				//Oś 1 staneła
				IF bRun1 AND ABS(Screwing1AxisRef.NcToPlc.ActVelo) < 150 THEN  //bylo 300
					mcHeightGearInMultiMaster.GearRatio1 	:=	0;
					mcHeightGearInMultiMaster.GearRatio2 	:=	lrSf2 * 	lrGearRatio2;
				END_IF
				//Oś 2 staneła		
				IF bRun2 AND ABS(Screwing2AxisRef.NcToPlc.ActVelo) < 150 THEN //bylo 300
					mcHeightGearInMultiMaster.GearRatio1 	:=	lrSf1 * 	lrGearRatio1;	
					mcHeightGearInMultiMaster.GearRatio2 	:=	0;				
				END_IF
				//Całkowite zatrzymanie - dwie osie staneły
				IF ABS(Screwing1AxisRef.NcToPlc.ActVelo) < 150 AND ABS(Screwing2AxisRef.NcToPlc.ActVelo) < 150 THEN //bylo 300
					mcHeightGearInMultiMaster.GearRatio1 	:=	0;
					mcHeightGearInMultiMaster.GearRatio2 	:=	0;	
				END_IF
				
				IF NOT bOptionMomentaryMode THEN	
					Running6ScrewingPositionTorqueMode();
				ELSE
					Running6ScrewingMomentaryMode();								
				END_IF
			END_IF
//====================================

	(*Przytrzymanie / Czas na odbpuszczenie chwytakow*)					
	E_GripperScrewer.eHolding:
		bGripper1Actuator				:=	FALSE;
		bGripper2Actuator				:=	FALSE;		
		IF tonGripper1ReliseDelay.Q AND tonGripper2ReliseDelay.Q THEN // Czas na otwarcie chwytaków
			IF tonHoldingTimer.Q OR NOT bOptionCapPushingWithoutScrewing THEN // Jeżeli jest włączona opcja wbijaka to czekaj na czas
				uiScrewing1TorqueControl	:=	0;
				uiScrewing2TorqueControl	:=	0;
				eRunningState				:=	E_GripperScrewer.eGoingUp;
			END_IF
		END_IF
	
//====================================	

	(*Podnoszenie do góry / reset laga i obrót do pozycji gotowości*)			 
	E_GripperScrewer.eGoingUp:
	
			CASE iGoingUpCase OF
				0:		
					mcScrewer1Stop.Execute					:=	FALSE;
					uiScrewing1TorqueControl				:=	0;	 					
					mcScrewer1SoftReset.Execute				:= FALSE;

					mcScrewer2Stop.Execute					:=	FALSE;
					uiScrewing2TorqueControl				:=	0;					
					mcScrewer2SoftReset.Execute				:= FALSE;			
					iGoingUpCase					:=	iGoingUpCase + 10;
		
				10: //Podjazd do góry i reset laga


					IF tonDelayBeforeResetLag.Q THEN//Reset laga
						mcScrewer1SoftReset.Execute	:= bRun1;
						mcScrewer2SoftReset.Execute	:= bRun2;
					END_IF
					//Sprawdzanie czy lag się zresetował
				IF	(mcScrewer1SoftReset.Done OR NOT bRun1) AND
					(mcScrewer2SoftReset.Done OR NOT bRun2) 
					(*AND	mcHeightMoveAbsolute.Done*)  THEN
						mcScrewer1SoftReset.Execute	:= FALSE;
						mcScrewer2SoftReset.Execute	:= FALSE;
						//mcHeightMoveAbsolute.Execute		:=	FALSE;
						iGoingUpCase				:= iGoingUpCase	+	10;					
					END_IF
				20:
				
					(*Przypisania dla ułatwienia*)
					lrDivider		:= 360.0/2;			
					CASE iMStep OF
						
						0: // Czy tu nie trzeba zrobić 
							iMStep							:= iMStep + 10;
							
						10: // Obliczanie najkrótszej pozycji, zależnie od ilość ramion chwytaka
							uiScrewing1TorqueControl		:= 6000; // Ustawianie momentu bo moze byc 0
							uiScrewing2TorqueControl		:= 6000; // Ustawianie momentu bo moze byc 0
					
							IF Screwing1AxisRef.NcToPlc.ActPos	>	0 THEN 	//Jeżeli aktualna pozycja jest >0 //w
								IF LMOD(Screwing1AxisRef.NcToPlc.ActPos,lrDivider)>(lrDivider/2) THEN // Dobieranie pozycji, tak żeby było bliżej
									mcScrewer1MoveAbsolute.Position		:=	Screwing1AxisRef.NcToPlc.ActPos+lrDivider			-	LMOD(Screwing1AxisRef.NcToPlc.ActPos,lrDivider);
								ELSE
									mcScrewer1MoveAbsolute.Position		:=	Screwing1AxisRef.NcToPlc.ActPos						-	LMOD(Screwing1AxisRef.NcToPlc.ActPos,lrDivider);			
								END_IF
							ELSE 							//Jezeli aktualna mniejsza od 0
								IF LMOD(ABS(Screwing1AxisRef.NcToPlc.ActPos),lrDivider)>(lrDivider/2) THEN // Dobieranie pozycji, tak żeby było bliżej
									mcScrewer1MoveAbsolute.Position		:=	Screwing1AxisRef.NcToPlc.ActPos-lrDivider			-	LMOD(Screwing1AxisRef.NcToPlc.ActPos,lrDivider);
								ELSE
									mcScrewer1MoveAbsolute.Position		:=	Screwing1AxisRef.NcToPlc.ActPos						-	LMOD(Screwing1AxisRef.NcToPlc.ActPos,lrDivider);		
								END_IF
							END_IF
							IF Screwing2AxisRef.NcToPlc.ActPos	>	0 THEN 	//Jeżeli aktualna pozycja jest >0 //w
								IF LMOD(Screwing2AxisRef.NcToPlc.ActPos,lrDivider)>(lrDivider/2) THEN // Dobieranie pozycji, tak żeby było bliżej
									mcScrewer2MoveAbsolute.Position		:=	Screwing2AxisRef.NcToPlc.ActPos+lrDivider			-	LMOD(Screwing2AxisRef.NcToPlc.ActPos,lrDivider);
								ELSE
									mcScrewer2MoveAbsolute.Position		:=	Screwing2AxisRef.NcToPlc.ActPos						-	LMOD(Screwing2AxisRef.NcToPlc.ActPos,lrDivider);			
								END_IF
							ELSE 							//Jezeli aktualna mniejsza od 0
								IF LMOD(ABS(Screwing2AxisRef.NcToPlc.ActPos),lrDivider)>(lrDivider/2) THEN // Dobieranie pozycji, tak żeby było bliżej
									mcScrewer2MoveAbsolute.Position		:=	Screwing2AxisRef.NcToPlc.ActPos-lrDivider			-	LMOD(Screwing2AxisRef.NcToPlc.ActPos,lrDivider);
								ELSE
									mcScrewer2MoveAbsolute.Position		:=	Screwing2AxisRef.NcToPlc.ActPos						-	LMOD(Screwing2AxisRef.NcToPlc.ActPos,lrDivider);		
								END_IF
							END_IF						
						
							iMStep						:= iMStep + 10;
					
						20: //Ruch
							mcScrewer1MoveAbsolute.Execute			:=	bEnable1;
							mcScrewer2MoveAbsolute.Execute			:=	bEnable2;		
							
							mcHeightMoveAbsolute.Position			:=	lrHeightReadyPosition;
							mcHeightMoveAbsolute.Velocity			:=	lrHeightSpeed;
							mcHeightMoveAbsolute.Execute			:=	TRUE;
							mcHeightMoveAbsolute.Execute			:=	TRUE;

							iMStep									:= iMStep + 10;	
						
						30: //Wykonano
							IF (mcScrewer1MoveAbsolute.Done OR NOT bRun1) AND	(mcScrewer2MoveAbsolute.Done OR NOT bRun2)    AND 
								mcHeightMoveAbsolute.Done
							THEN
								mcScrewer1MoveAbsolute.Execute		:=	FALSE;
								mcScrewer2MoveAbsolute.Execute		:=	FALSE;
								mcHeightMoveAbsolute.Execute		:=	FALSE;
								iMStep							:= 100;			
							END_IF
							
						100: //Koniec
							iMStep						:= 0;
							iGoingUpCase					:= iGoingUpCase	+	20;	
					END_CASE
								
				40:	//Koniec
					eRunningState								:= E_GripperScrewer.eDone;
					iGoingUpCase						:= 0;		
			END_CASE
		
//====================================			
	(*Zakręcono*)			
	E_GripperScrewer.eDone:
	
		rScrewing1ProportionalGain			:= 10;
		rScrewing2ProportionalGain			:= 10;
	
		bScrewed1							:=	FALSE;
		bScrew1Found						:=	FALSE;
		bScrewed2							:=	FALSE;
		bScrew2Found						:=	FALSE;
		
		mcScrewer1Stop.Execute				:=	FALSE;
		mcScrewer2Stop.Execute				:=	FALSE;		
	
		mcHeightStop.Execute				:=	FALSE;
		bCycleDone1 						:=	NOT bWarning1 AND bRun1;
		bCycleNotDone1						:=	bWarning1 OR NOT bRun1;
		bCycleDone2 						:=	NOT bWarning2 AND bRun2;
		bCycleNotDone2						:=	bWarning2 OR NOT bRun2;		
		
		eRunningState 						:=	E_GripperScrewer.eReady;	

//====================================	
			
	E_GripperScrewer.eNotDone:
	
		bCycleNotDone1 						:=	TRUE;
		bCycleNotDone2						:=	TRUE;
		eRunningState						:=	E_GripperScrewer.eReady;	
		mcScrewer1SoftReset					(Axis:=Screwing1AxisRef, Execute:=bRun1);
		mcScrewer2SoftReset					(Axis:=Screwing2AxisRef, Execute:=bRun2);	
	
END_CASE
END_ACTION

ACTION Running2ToPushingPosition:
		(*w2*)
		CASE iToPushingPositionCASE OF 
			
		0:(*0*)
			bGripper1Actuator									:=	FALSE;
			bGripper2Actuator									:=	FALSE;
			iToPushingPositionCASE								:=	iToPushingPositionCASE	+	10;
			
		10:(*Start*)
			mcHeightMoveAbsolute.Execute						:=	TRUE;
			mcHeightMoveAbsolute.Velocity						:=	lrHeightSpeed;
			mcHeightMoveAbsolute.Position						:=	lrHeightPushingPosition;
			iToPushingPositionCASE								:=	iToPushingPositionCASE	+	10;		
			
		20:(*Opcja - obrót do tyłu w momencie dojazdu do pozycji docisku*)
			IF bOptionScrewingBackwardsInPushingPosition THEN
				lrFindigScrewDegree								:=	360;	
				                                				
				uiScrewing1TorqueControl						:=	6000;
				mcScrewer1MoveRelative.Velocity					:=	lrScrewerSpeed/2;		
				mcScrewer1MoveRelative.Execute					:=	bRun1;
				                                				
				uiScrewing2TorqueControl						:=	6000;
				mcScrewer2MoveRelative.Velocity					:=	lrScrewerSpeed/2;		
				mcScrewer2MoveRelative.Execute					:=	bRun2;
				iToPushingPositionCASE							:=	iToPushingPositionCASE	+	10;
			ELSE
				iToPushingPositionCASE							:=	iToPushingPositionCASE	+	10;
			END_IF                                          	

(*		30: (*Spr.*)
			IF mcHeightMoveAbsolute.Done AND
				(mcScrewer1MoveRelative.Done OR NOT bOptionScrewingBackwardsInPushingPosition OR NOT bRun1) AND 	
				(mcScrewer2MoveRelative.Done OR NOT bOptionScrewingBackwardsInPushingPosition OR NOT bRun2) 	 			
			THEN	
				mcHeightMoveAbsolute.Execute					:=	FALSE;
				mcScrewer1MoveRelative.Execute					:=	FALSE;
				mcScrewer2MoveRelative.Execute					:=	FALSE;	
				iToPushingPositionCASE							:=	iToPushingPositionCASE	+	10;
			END_IF*)
			
		30: (*Spr.*)
			IF iTool = 4 THEN
				IF mcHeightMoveAbsolute.Done 	 			
				THEN	
					mcHeightMoveAbsolute.Execute					:=	FALSE;
					mcScrewer1MoveRelative.Execute					:=	FALSE;
					mcScrewer2MoveRelative.Execute					:=	FALSE;	
					iToPushingPositionCASE							:=	iToPushingPositionCASE	+	10;
				END_IF	
			ELSE
				IF mcHeightMoveAbsolute.Done AND
				(mcScrewer1MoveRelative.Done OR NOT bOptionScrewingBackwardsInPushingPosition OR NOT bRun1) AND 	
				(mcScrewer2MoveRelative.Done OR NOT bOptionScrewingBackwardsInPushingPosition OR NOT bRun2) 	 			
				THEN	
					mcHeightMoveAbsolute.Execute					:=	FALSE;
					mcScrewer1MoveRelative.Execute					:=	FALSE;
					mcScrewer2MoveRelative.Execute					:=	FALSE;	
					iToPushingPositionCASE							:=	iToPushingPositionCASE	+	10;
				END_IF
			END_IF
		40:  (*Opcja - Dodatkowe zamknięcie chwytakiem przed zakręceniem *)
				IF bOptionCapPositioning AND sTool <> 'ksztaltowa/do kulek' AND sTool <> 'wbijajaca' THEN
					CASE iCloseGripperBeforeScrewingCASE OF
						0:
							bGripper1Actuator					:=	bRun1;
							bGripper2Actuator					:=	bRun2;
							iCloseGripperBeforeScrewingCASE		:=	iCloseGripperBeforeScrewingCASE	+10;
						10:	
							IF 	(tonGripper1Delay.Q OR NOT bRun1) AND 
								(tonGripper2Delay.Q OR NOT bRun2) 
							THEN					
								iCloseGripperBeforeScrewingCASE	:=	iCloseGripperBeforeScrewingCASE	+10;
							END_IF
						20:	
								bGripper1Actuator				:=	bGripper1Actuator	:=	FALSE;		
								iCloseGripperBeforeScrewingCASE	:=	iCloseGripperBeforeScrewingCASE	+10;
						30:
							IF 	(tonGripper1ReliseDelay2.Q OR NOT bRun1) AND 
								(tonGripper2ReliseDelay2.Q OR NOT bRun2) 
							THEN					
								iCloseGripperBeforeScrewingCASE	:=	iCloseGripperBeforeScrewingCASE	+10;
							END_IF
						40:
						
							iCloseGripperBeforeScrewingCASE		:=	0;
							iToPushingPositionCASE				:=	iToPushingPositionCASE	+	10;							
					END_CASE
				ELSE
					iToPushingPositionCASE						:=	iToPushingPositionCASE	+	10;
				END_IF

			
		50:	 (*Zamkniecie chwytaka i przejazd dalej*)
			IF sTool <> 'ksztaltowa/do kulek' AND sTool <> 'wbijajaca' THEN
				bGripper1Actuator								:=	bRun1;
				bGripper2Actuator								:=	bRun2;
			ELSE                                    	
				bGripper1Actuator								:=	FALSE;
				bGripper2Actuator								:=	FALSE;
			END_IF	

			IF bOptionOpenedGripperWhenFindingScrew AND bOptionFindScrewInPushingPosition THEN
				bGripper1Actuator								:=	FALSE;
				bGripper2Actuator								:=	FALSE;
			END_IF
			
			IF 	(tonGripper1Delay.Q OR sTool = 'ksztaltowa/do kulek' OR sTool = 'wbijajaca' OR bOptionOpenedGripperWhenFindingScrew AND bOptionFindScrewInPushingPosition OR NOT bRun1) AND 
				(tonGripper2Delay.Q OR sTool = 'ksztaltowa/do kulek' OR sTool = 'wbijajaca' OR bOptionOpenedGripperWhenFindingScrew AND bOptionFindScrewInPushingPosition OR NOT bRun2) 
			THEN
          		         	
				iToPushingPositionCASE							:=	iToPushingPositionCASE	+	10;
			END_IF	
		
				
		60:(*Opcja - Obrót z pozycji docisku do zakrecania *)
			IF bOptionFindScrewRotateFromPushingToScrewingSensor AND NOT bOptionFindScrewInPushingPosition THEN
				lrFindigScrewDegree								:=	180;	
			                                    				
				uiScrewing1TorqueControl						:=	6000;
				mcScrewer1MoveRelative.Velocity					:=	lrScrewerSpeed*1.5;	//sky is the limit - nie wiadomo po co to robimy 	
				mcScrewer1MoveRelative.Execute					:=	bRun1;
							                    				
				uiScrewing2TorqueControl						:=	6000;
				mcScrewer2MoveRelative.Velocity					:=	lrScrewerSpeed*1.5;		
				mcScrewer2MoveRelative.Execute					:=	bRun2;
				iToPushingPositionCASE							:=	iToPushingPositionCASE	+	10;
				
			ELSE 
				iToPushingPositionCASE							:=	iToPushingPositionCASE	+	10;
			END_IF
			
		70: //Dodatkowy ruch do góry tylko dla głowicy zasysającej // DO USUNIECIA 
			IF iTool = 4 THEN
				mcHeightMoveAbsolute.Execute						:=	TRUE; // DO USUNIECIA 
				mcHeightMoveAbsolute.Velocity						:=	lrHeightSpeed; // DO USUNIECIA 
				mcHeightMoveAbsolute.Position						:=	lrHeightPushingPosition+50; // DO USUNIECIA 
				IF mcHeightMoveAbsolute.Done THEN // DO USUNIECIA 
					mcScrewer1Stop.Execute 							:= bRun1;
					mcScrewer2Stop.Execute 							:= bRun2;					
					mcHeightMoveAbsolute.Execute					:=	FALSE;; // DO USUNIECIA 
					iToPushingPositionCASE							:=	iToPushingPositionCASE	+	10;		 // DO USUNIECIA 	
				END_IF // DO USUNIECIA 
			ELSE
				iToPushingPositionCASE							:=	iToPushingPositionCASE	+	10;		 // DO USUNIECIA 	
			END_IF
		80: // DO ZMIANY NA 70
			//tutaj bym dodał warunek od ugięcia sprężyny, bo to jedyna rzecz która jest progresywna + zatrzymanie zakręcarki 

			IF 	(mcScrewer1Stop.Done OR (NOT bOptionScrewingBackwardsInPushingPosition OR bOptionFindScrewRotateFromPushingToScrewingSensor) OR NOT bRun1) AND 	
				(mcScrewer2Stop.Done OR (NOT bOptionScrewingBackwardsInPushingPosition OR bOptionFindScrewRotateFromPushingToScrewingSensor) OR NOT bRun2) 
			THEN
				mcScrewer1Stop.Execute	:= FALSE;
				mcScrewer2Stop.Execute	:= FALSE;		
				IF bOptionFindScrewInPushingPosition THEN
					eRunningState									:=	E_GripperScrewer.eFindingScrew;
				ELSE
					eRunningState									:=	E_GripperScrewer.eToScrewingPosition;
				END_IF
				
				iToPushingPositionCASE						:=	0;
			END_IF
				
		END_CASE
END_ACTION

ACTION Running5FindingScrew:
(*Opcja 1 Szukania gwintu - zwykłe szukanie*) 
IF NOT bOptionFindScrewWithHeightSensor THEN
	(*Opcja cofniecie o zadany kąt*)	
	CASE iFindingScrewCASE OF
				
			0:	// Czyszczenie
				mcScrewer1MoveRelative.Execute				:=	FALSE;
				mcScrewer2MoveRelative.Execute				:=	FALSE;		
				lrScrewer1MaxTorqueWhenFindingScrew			:=	0;
				lrScrewer2MaxTorqueWhenFindingScrew			:=	0;
				lrStartPosition1FindingScrew 				:=	Screwing1AxisRef.NcToPlc.ActPos;
				lrStartPosition2FindingScrew 				:=	Screwing2AxisRef.NcToPlc.ActPos;			
				uiScrewing1TorqueControl					:=	6000;
				uiScrewing2TorqueControl					:=	6000;			
				bScrew1Found								:=	FALSE;
				bScrew2Found								:=	FALSE;
				iFindingScrewCASE							:=	iFindingScrewCASE	+	10;
						
			10: (*ruch o zadany kat*)
				mcScrewer1MoveRelative.Velocity		:=	lrScrewerSpeed;
				mcScrewer1MoveRelative.Execute		:=	bRun1;
				
				mcScrewer2MoveRelative.Velocity		:=	lrScrewerSpeed;
				mcScrewer2MoveRelative.Execute		:=	bRun2;
				
				IF	(NOT bRun1 OR mcScrewer1MoveRelative.Done) AND
					(NOT bRun2 OR mcScrewer2MoveRelative.Done)
			
				THEN		
					lrScrewer1MaxTorqueWhenFindingScrew	:= 0;
					lrScrewer2MaxTorqueWhenFindingScrew	:= 0;
					mcScrewer1MoveRelative.Execute		:=	FALSE;
					mcScrewer1MoveRelative.Execute		:=	FALSE;
					iFindingScrewCASE					:=	iFindingScrewCASE	+	10;	
				END_IF
					
			20:
				lrStartPosition1						:=	Screwing1AxisRef.NcToPlc.ActPos;
				lrStartPosition2						:=	Screwing2AxisRef.NcToPlc.ActPos;
				iFindingScrewCASE 						:=	0;
				eRunningState							:=	E_GripperScrewer.eScrewing;
				IF bOptionFindScrewInPushingPosition THEN // Opcja - szukanie gwintu w pozycji docisku
					// Przejście do pozycji zakręcania, dlatego że był w pozycji docisku
					eRunningState							:=	E_GripperScrewer.eToScrewingPosition;
				END_IF
				IF NOT bHeightGearingWithScrewer THEN 	(* Wersja bez gearowania*)
					mcScrewer1MoveVelocity.Execute		:= bRun1;
					mcScrewer2MoveVelocity.Execute		:= bRun2;
					eRunningState:=E_GripperScrewer.eScrewing;
				ELSE 									(* Wersja z gearowaniem*)
					iFindingScrewCASE 						:=	0;
					eRunningState							:=	E_GripperScrewer.eScrewing;
					IF bOptionFindScrewInPushingPosition THEN // Opcja - szukanie gwintu w pozycji docisku
						// Przejście do pozycji zakręcania, dlatego że był w pozycji docisku
						eRunningState							:=	E_GripperScrewer.eToScrewingPosition;
					END_IF
				END_IF
	END_CASE

ELSE 
(*	(*Opcja 2 Szukania gwintu - szukanie z czujnikiem wysokości*) 
		CASE iFindingScrewCASE OF
			
		0:	// Czyszczenie
			mcScrewer1MoveRelative.Execute				:=	FALSE;
			//lrScrewerMaxSensorHeightWhenFindingScrew	:=	-100000; //Musi być INIT -100000
			//lrScrewerMinSensorHeightWhenFindingScrew	:=	0;
			lrStartPosition1FindingScrew 				:=	Screwing1AxisRef.NcToPlc.ActPos;
			lrStartPosition2FindingScrew 				:=	Screwing2AxisRef.NcToPlc.ActPos;			
			uiScrewing1TorqueControl					:=	6000;
			uiScrewing2TorqueControl					:=	6000;			
			bScrew1Found								:=	FALSE;
			bScrew2Found								:=	FALSE;
			bScrew1MinFound								:=	FALSE;
			bScrew2MinFound								:=	FALSE;			
			iFindingScrewCASE							:=	iFindingScrewCASE	+	10;
			// Skasuj wartości jeżeli ponownie włączono szukanie wysokości
			IF bFindScrewAdjustSensorHeight THEN
				lrScrewerMaxSensorHeightWhenFindingScrew	:=	-100000; //Musi być INIT -100000
				lrScrewerMinSensorHeightWhenFindingScrew	:=	100000;
			END_IF
			
		10: // Rozpoczęcie ruchu w tył i szukanie MIN i MAX momentu
			// Tylko 1 zakręcarka szuka Min i Max po każdej zmianie
			// Uruchom szukanie jeżeli są wartości domyślne
			IF lrScrewerMaxSensorHeightWhenFindingScrew = -100000 OR lrScrewerMinSensorHeightWhenFindingScrew = 100000 THEN
				bFindScrewAdjustSensorHeight				:= TRUE;
				lrScrewerMaxSensorHeightWhenFindingScrew	:=	-100000; //Musi być INIT -100000
				lrScrewerMinSensorHeightWhenFindingScrew	:=	100000;
			END_IF
			
			IF bFindScrewAdjustSensorHeight THEN
				uiScrewing1TorqueControl					:=	6000;
				lrFindigScrewDegree							:=	720;
				mcScrewer1MoveRelative.Velocity				:=	200;
				mcScrewer1MoveRelative.Execute				:=	bRun1;
							
				IF lrScrewerMaxSensorHeightWhenFindingScrew<diSensorHeightCV THEN
					lrScrewerMaxSensorHeightWhenFindingScrew:=	diSensorHeightCV;
				END_IF			
				IF lrScrewerMinSensorHeightWhenFindingScrew>diSensorHeightCV THEN
					lrScrewerMinSensorHeightWhenFindingScrew:=	diSensorHeightCV;
				END_IF		
			
				IF (mcScrewer1MoveRelative.Done OR NOT bRun1) THEN
					mcScrewer1MoveRelative.Execute			:=	FALSE;
					bFindScrewAdjustSensorHeight			:=	FALSE;	iFindScrewAdjustSensorHeight	:=	iFindScrewAdjustSensorHeight	+	1;
					iFindingScrewCASE						:=	iFindingScrewCASE	+	10;
				END_IF
			ELSE
				iFindingScrewCASE						:=	iFindingScrewCASE	+	10;
			END_IF

		20: // (Nie potrzebne) Przejście dalej gdy jest gotowość
			IF NOT mcScrewer1MoveRelative.Busy AND NOT mcScrewer2MoveRelative.Busy THEN
				lrStartPosition1FindingScrew 			:=	Screwing1AxisRef.NcToPlc.ActPos;
				lrStartPosition2FindingScrew 			:=	Screwing2AxisRef.NcToPlc.ActPos;				
				iFindingScrewCASE						:=	iFindingScrewCASE	+	10;				
			END_IF
			
		30: // Rozpoczęcie szukanie największego momentu o określony maksymalny kąt
			uiScrewing1TorqueControl					:=	6000;
			mcScrewer1MoveRelative.Velocity				:=	500;//lrScrewerSpeed;///2;
			mcScrewer1MoveRelative.Execute				:=	bRun1;
			
			uiScrewing2TorqueControl					:=	6000;
			mcScrewer2MoveRelative.Velocity				:=	500;//lrScrewerSpeed;///2;
			mcScrewer2MoveRelative.Execute				:=	bRun2;		
	
			iFindingScrewCASE							:=	iFindingScrewCASE	+	10;	
			
		40:	//Szukanie określonego momentu po 200 st. i zatrzymanie ruchu 

			(*Pierwsze szukanie*)
			IF NOT bScrew1MinFound THEN															(*W1*)
				IF ABS(ABS(lrStartPosition1FindingScrew)-ABS(Screwing1AxisRef.NcToPlc.ActPos))	>	100  THEN 
					IF diSensorHeightCV < ((lrScrewerMaxSensorHeightWhenFindingScrew+lrScrewerMinSensorHeightWhenFindingScrew)/2) THEN		(*W2*) //Dla Słoików 300ml						
						bScrew1MinFound						:=	TRUE;
						lrStartPosition1FindingScrew 		:=	Screwing1AxisRef.NcToPlc.ActPos;
					END_IF	
				END_IF
			END_IF
			IF NOT bScrew2MinFound THEN															(*W1*)
				IF ABS(ABS(lrStartPosition2FindingScrew)-ABS(Screwing2AxisRef.NcToPlc.ActPos))	>	100  THEN 
					IF diSensorHeightCV < ((lrScrewerMaxSensorHeightWhenFindingScrew+lrScrewerMinSensorHeightWhenFindingScrew)/2) THEN		(*W2*)	//Dla Słoików 300ml	
						bScrew2MinFound						:=	TRUE;	
						lrStartPosition2FindingScrew 		:=	Screwing2AxisRef.NcToPlc.ActPos;
					END_IF	
				END_IF	
			END_IF
			lrScrewerOffsetSensorHeightWhenFindingScrew	:=	((lrScrewerMaxSensorHeightWhenFindingScrew+lrScrewerMinSensorHeightWhenFindingScrew)/2)
																+(lrScrewerMinSensorHeightWhenFindingScrew-lrScrewerMaxSensorHeightWhenFindingScrew)/6;
			
			(*Drugie szukanie*)																					(*W3*)
			IF bScrew1MinFound AND ABS(ABS(lrStartPosition1FindingScrew)-ABS(Screwing1AxisRef.NcToPlc.ActPos))	>	10  THEN 
				IF diSensorHeightCV > lrScrewerOffsetSensorHeightWhenFindingScrew THEN		(*W4*)	//Dla Słoików 300ml
					bScrew1Found						:=	TRUE;
					mcScrewer1MoveRelative.Execute		:=	FALSE;
					lrStartPosition1FindingScrew 		:=	Screwing1AxisRef.NcToPlc.ActPos;
				END_IF
			END_IF																								(*W3*)
			IF bScrew2MinFound AND ABS(ABS(lrStartPosition2FindingScrew)-ABS(Screwing2AxisRef.NcToPlc.ActPos))	>	10 THEN 
				IF diSensorHeightCV > ((lrScrewerMaxSensorHeightWhenFindingScrew+lrScrewerMinSensorHeightWhenFindingScrew)/2) THEN		(*W4*)	//Dla Słoików 300ml
					bScrew2Found						:=	TRUE;
					mcScrewer2MoveRelative.Execute		:=	FALSE;
					lrStartPosition2FindingScrew 		:=	Screwing1AxisRef.NcToPlc.ActPos;
				END_IF
			END_IF

			IF bScrew1Found  THEN
				uiScrewing1TorqueControl		:=	6000;
				mcScrewer1Stop.Execute			:=	TRUE;			
			END_IF
			
			IF bScrew2Found  THEN
				uiScrewing2TorqueControl		:=	6000;
				mcScrewer2Stop.Execute			:=	TRUE;
			END_IF			
			
			IF	((bScrew1Found AND mcScrewer1Stop.Done) OR NOT bRun1 OR mcScrewer1MoveRelative.Done) AND
				((bScrew2Found AND mcScrewer2Stop.Done) OR NOT bRun2 OR mcScrewer2MoveRelative.Done)
			THEN
				 mcScrewer1MoveRelative.Execute 	:=	FALSE;
				 mcScrewer1Stop.Execute				:=	FALSE;
				 mcScrewer2MoveRelative.Execute 	:=	FALSE;		
				 mcScrewer2Stop.Execute				:=	FALSE;	 
				 iFindingScrewCASE					:=	iFindingScrewCASE	+	10;	
			END_IF
			
		50: 
			IF tonFindingScrewDelay.Q THEN
 				iFindingScrewCASE					:=	iFindingScrewCASE	+	10;						
			END_IF


		60:
			lrStartPosition1						:=	Screwing1AxisRef.NcToPlc.ActPos;
			lrStartPosition2						:=	Screwing2AxisRef.NcToPlc.ActPos;
			iFindingScrewCASE 						:=	0;
			eRunningState							:=	E_GripperScrewer.eScrewing;
			IF bOptionFindScrewInPushingPosition THEN // Opcja - szukanie gwintu w pozycji docisku
				// Przejście do pozycji zakręcania, dlatego że był w pozycji docisku
				eRunningState							:=	E_GripperScrewer.eToScrewingPosition;
			END_IF
		END_CASE *)
		
		(*Opcja 3 Szukania gwintu - szukanie z czujnikiem pod hindusa*) 
		CASE iFindingScrewCASE OF
			
		0:	// Czyszczenie
			mcScrewer1MoveRelative.Execute				:=	FALSE;
			lrStartPosition1FindingScrew 				:=	Screwing1AxisRef.NcToPlc.ActPos;
			lrStartPosition2FindingScrew 				:=	Screwing2AxisRef.NcToPlc.ActPos;			
			uiScrewing1TorqueControl					:=	6000;
			uiScrewing2TorqueControl					:=	6000;			
			bScrew1Found								:=	FALSE;
			bScrew2Found								:=	FALSE;
			bScrew1MinFound								:=	FALSE;
			bScrew2MinFound								:=	FALSE;			
			iFindingScrewCASE							:=	iFindingScrewCASE	+	10;
			lrScrewerMaxSensorHeightWhenFindingScrew	:=	-100000; //Musi być INIT -100000
			lrScrewerMinSensorHeightWhenFindingScrew	:=	100000;

			
		10: // Rozpoczęcie ruchu w tył i szukanie MIN i MAX momentu
			// Tylko 1 zakręcarka szuka Min i Max po każdej zmianie
			// Uruchom szukanie jeżeli są wartości domyślne
			IF lrScrewerMaxSensorHeightWhenFindingScrew = -100000 OR lrScrewerMinSensorHeightWhenFindingScrew = 100000 THEN
				bFindScrewAdjustSensorHeight				:= TRUE;
				lrScrewerMaxSensorHeightWhenFindingScrew	:=	-100000; //Musi być INIT -100000
				lrScrewerMinSensorHeightWhenFindingScrew	:=	100000;
			END_IF		
			iFindingScrewCASE							:=	iFindingScrewCASE	+	10;

		20: // (Nie potrzebne) Przejście dalej gdy jest gotowość
			IF NOT mcScrewer1MoveRelative.Busy AND NOT mcScrewer2MoveRelative.Busy THEN
				lrStartPosition1FindingScrew 			:=	Screwing1AxisRef.NcToPlc.ActPos;
				lrStartPosition2FindingScrew 			:=	Screwing2AxisRef.NcToPlc.ActPos;				
				iFindingScrewCASE						:=	iFindingScrewCASE	+	10;				
			END_IF
			
		30: // Rozpoczęcie szukanie największego momentu o określony maksymalny kąt
			uiScrewing1TorqueControl					:=	6000;
			mcScrewer1MoveRelative.Velocity				:=	lrScrewerSpeed;//1000;//500;//lrScrewerSpeed;///2;
			mcScrewer1MoveRelative.Execute				:=	bRun1;
			
			uiScrewing2TorqueControl					:=	6000;
			mcScrewer2MoveRelative.Velocity				:=	lrScrewerSpeed;//1000;//500;//lrScrewerSpeed;///2;
			mcScrewer2MoveRelative.Execute				:=	bRun2;		
	
			iFindingScrewCASE							:=	iFindingScrewCASE	+	10;	
			
		40:	//Szukanie określonego momentu po 200 st. i zatrzymanie ruchu 

			IF ABS(ABS(lrStartPosition1FindingScrew)-ABS(Screwing1AxisRef.NcToPlc.ActPos))	>	50 THEN			(* KROK 1 - ROZPEDZENIE 50st. - po 50st. szukanie max i min*)
				IF lrScrewerMaxSensorHeightWhenFindingScrew<lrSpringHeightCV THEN
					lrScrewerMaxSensorHeightWhenFindingScrew:=	lrSpringHeightCV;
				END_IF			
				IF lrScrewerMinSensorHeightWhenFindingScrew>lrSpringHeightCV THEN
					lrScrewerMinSensorHeightWhenFindingScrew:=	lrSpringHeightCV;
				END_IF	
			END_IF
		
			(*Pierwsze szukanie*)
			IF NOT bScrew1MinFound THEN														
				IF ABS(ABS(lrStartPosition1FindingScrew)-ABS(Screwing1AxisRef.NcToPlc.ActPos))	>	100  THEN 	(* KROK 2 - PIERWSZY SKOK 100st. - po 100st. szukanie spadku o 0,5mm*)
					IF lrSpringHeightCV < (lrScrewerMaxSensorHeightWhenFindingScrew-0.5) THEN	//0,5mm				
						bScrew1MinFound								:=	TRUE;
						lrStartPosition1FindingScrew 				:=	Screwing1AxisRef.NcToPlc.ActPos;
						IF bScrew1MinFound THEN	{warning ' tutaj nie będzie działać dla dwóch zakręcarek na 1 podnosniku*)}
							lrScrewerMaxSensorHeightWhenFindingScrew	:=	-100000; //Musi być INIT -100000
							lrScrewerMinSensorHeightWhenFindingScrew	:=	100000;
						END_IF	
					END_IF	
				END_IF
			END_IF
			IF NOT bScrew2MinFound THEN															
				IF ABS(ABS(lrStartPosition2FindingScrew)-ABS(Screwing2AxisRef.NcToPlc.ActPos))	>	100  THEN 	
					IF lrSpringHeightCV < (lrScrewerMaxSensorHeightWhenFindingScrew-0.5) THEN	//0,5mm
						bScrew2MinFound						:=	TRUE;	
						lrStartPosition2FindingScrew 		:=	Screwing2AxisRef.NcToPlc.ActPos;
					END_IF	
				END_IF	
			END_IF

			(*Drugie szukanie*)																				
			IF bScrew1MinFound AND ABS(ABS(lrStartPosition1FindingScrew)-ABS(Screwing1AxisRef.NcToPlc.ActPos))	>	100  THEN 	(* KROK 3 - DRUGI SKOK 100st. - po 100st. szukanie spadku o 0,5mm*)			
				IF lrSpringHeightCV < (lrScrewerMaxSensorHeightWhenFindingScrew-0.5) THEN	//0,5mm
					bScrew1Found						:=	TRUE;
					mcScrewer1MoveRelative.Execute		:=	FALSE;
					lrStartPosition1FindingScrew 		:=	Screwing1AxisRef.NcToPlc.ActPos;
				END_IF
			END_IF																							
			IF bScrew2MinFound AND ABS(ABS(lrStartPosition2FindingScrew)-ABS(Screwing2AxisRef.NcToPlc.ActPos))	>	100 THEN 
				IF lrSpringHeightCV < (lrScrewerMaxSensorHeightWhenFindingScrew-0.5)  THEN	//0,5mm	
					bScrew2Found						:=	TRUE;
					mcScrewer2MoveRelative.Execute		:=	FALSE;
					lrStartPosition2FindingScrew 		:=	Screwing2AxisRef.NcToPlc.ActPos;
				END_IF
			END_IF

			IF 		lrPackageThreadTimes 	<= 1 OR lrPackageThreadTimes >= 4 	THEN lrFindingScrewPositionDelay := 30; 
			ELSIF 	lrPackageThreadTimes 	= 2 								THEN lrFindingScrewPositionDelay := 90;			
			ELSIF	lrPackageThreadTimes 	= 3 								THEN lrFindingScrewPositionDelay := 60; END_IF
			
			IF (bScrew1Found OR (bScrew1MinFound AND lrPackageThreadTimes = 1)) AND ABS(ABS(lrStartPosition1FindingScrew)-ABS(Screwing1AxisRef.NcToPlc.ActPos))	> lrFindingScrewPositionDelay THEN	(* KROK 4 - PRZEJAZD - przejazd o 30st po druch skokach*)
				uiScrewing1TorqueControl		:=	6000;
				mcScrewer1Stop.Execute			:=	TRUE;				
			END_IF
			
			IF (bScrew2Found OR (bScrew2MinFound AND lrPackageThreadTimes = 1)) AND ABS(ABS(lrStartPosition2FindingScrew)-ABS(Screwing2AxisRef.NcToPlc.ActPos))	> lrFindingScrewPositionDelay THEN
				uiScrewing2TorqueControl		:=	6000;
				mcScrewer2Stop.Execute			:=	TRUE;
			END_IF			
			
			IF	(((bScrew1Found OR (bScrew1MinFound AND lrPackageThreadTimes = 1)) AND mcScrewer1Stop.Done) OR NOT bRun1 OR mcScrewer1MoveRelative.Done) AND
				(((bScrew2Found OR (bScrew2MinFound AND lrPackageThreadTimes = 1)) AND mcScrewer2Stop.Done) OR NOT bRun2 OR mcScrewer2MoveRelative.Done)
			THEN
				 mcScrewer1MoveRelative.Execute 	:=	FALSE;
				 mcScrewer1Stop.Execute				:=	FALSE;
				 mcScrewer2MoveRelative.Execute 	:=	FALSE;		
				 mcScrewer2Stop.Execute				:=	FALSE;	 
				 iFindingScrewCASE					:=	iFindingScrewCASE	+	10;	
			END_IF
			
		50: 
			IF tonFindingScrewDelay.Q THEN
 				iFindingScrewCASE					:=	iFindingScrewCASE	+	10;						
			END_IF

		60:
			lrStartPosition1						:=	Screwing1AxisRef.NcToPlc.ActPos;
			lrStartPosition2						:=	Screwing2AxisRef.NcToPlc.ActPos;
			iFindingScrewCASE 						:=	0;
			eRunningState							:=	E_GripperScrewer.eScrewing;
			IF bOptionFindScrewInPushingPosition THEN // Opcja - szukanie gwintu w pozycji docisku
				// Przejście do pozycji zakręcania, dlatego że był w pozycji docisku
				eRunningState							:=	E_GripperScrewer.eToScrewingPosition;
			END_IF
		END_CASE
END_IF
END_ACTION

ACTION Running6ScrewingMomentaryMode:
				(********** TRYB MOMENTOWY **********)
					CASE iScrewingCase OF 	
					0:
						(* Wersja 2 - gearowanie Multi Master***************************************************************) 
						IF iTool <> 2 THEN
							bGripper1Actuator						:=	bRun1; // Ponowne załączanie chwytaków, dlatego
							bGripper2Actuator						:=	bRun2; // że jest możliwa duża ilość opcji
						ELSE
							bGripper1Actuator						:=	FALSE; // Ponowne załączanie chwytaków, dlatego
							bGripper2Actuator						:=	FALSE;
						END_IF
						mcHeightGearInMultiMaster.Enable			:=	TRUE;				
						(* Start zakręcania *)
						IF	mcHeightGearInMultiMaster.InGear AND 
							(tonGripper1Delay.Q OR sTool = 'ksztaltowa/do kulek' OR NOT bRun1) AND (tonGripper2Delay.Q OR sTool = 'ksztaltowa/do kulek'  OR NOT bRun2) // ton'y powinny być już wczesniej załączone jeżeli były chwytaki	
						THEN

							mcScrewer1TorqueControl.Execute					:=	bRun1;
							mcScrewer1TorqueControl.Torque					:=	5000;//(INT_TO_UINT(iScrewer1SetTorque+3)*10)+iScrewer1AddTorque;	
							mcScrewer1TorqueControl.TorqueRamp				:=	4000;
							mcScrewer1TorqueControl.VelocityLimitHigh		:=	10;							
							mcScrewer1TorqueControl.VelocityLimitLow		:=	-5000;//(lrScrewerSpeed);
												
							mcScrewer2TorqueControl.Execute					:=	bRun2;
							mcScrewer2TorqueControl.Torque					:=	5000;//(INT_TO_UINT(iScrewer2SetTorque+3)*10)+iScrewer2AddTorque;	
							mcScrewer2TorqueControl.TorqueRamp				:=	4000;
							mcScrewer2TorqueControl.VelocityLimitHigh		:=	10;							
							mcScrewer2TorqueControl.VelocityLimitLow		:=	-5000;//(lrScrewerSpeed);
	
							iScrewingCase									:=	iScrewingCase + 10;			
						END_IF
						
					10:	
					
						IF ABS(ABS(lrStartPosition1)-ABS(Screwing1AxisRef.NcToPlc.ActPos))>(lrPackageTurnoversToFullScrewed*360.0/7)  THEN 
							mcScrewer1TorqueControl.Torque					:=	-9;		
							mcScrewer1TorqueControl.TorqueRamp				:=	1500;					
							mcScrewer1TorqueControl.VelocityLimitLow		:=	-4000;
						END_IF	
							
						IF ABS(ABS(lrStartPosition2)-ABS(Screwing2AxisRef.NcToPlc.ActPos))>(lrPackageTurnoversToFullScrewed*360.0/7)  THEN 
							mcScrewer2TorqueControl.Torque					:=	-9;		
							mcScrewer2TorqueControl.TorqueRamp				:=	1500;					
							mcScrewer2TorqueControl.VelocityLimitLow		:=	-4000;
						END_IF	
						
						IF ABS(ABS(lrStartPosition1)-ABS(Screwing1AxisRef.NcToPlc.ActPos))>(lrPackageTurnoversToFullScrewed*360.0/6)  THEN 
							mcScrewer1TorqueControl.Torque					:=	(INT_TO_UINT(iScrewer1SetTorque)+iScrewer1AddTorque);		
							mcScrewer1TorqueControl.TorqueRamp				:=	4000;					
							mcScrewer1TorqueControl.VelocityLimitLow		:=	-(lrScrewerSpeed);
						END_IF	
							
						IF ABS(ABS(lrStartPosition2)-ABS(Screwing2AxisRef.NcToPlc.ActPos))>(lrPackageTurnoversToFullScrewed*360.0/6)  THEN 
							mcScrewer2TorqueControl.Torque					:=	(INT_TO_UINT(iScrewer2SetTorque)+iScrewer2AddTorque);		
							mcScrewer2TorqueControl.TorqueRamp				:=	4000;					
							mcScrewer2TorqueControl.VelocityLimitLow		:=	-(lrScrewerSpeed);
						END_IF						
						(*IF tonMomentaryScrewing1Timer.Q OR bWarning1 THEN
							mcScrewer1Stop.Execute				:=	TRUE;
							bGripper1Actuator					:=	FALSE;
							mcScrewer1TorqueControl.Execute		:=	FALSE;
							uiScrewing1TorqueControl			:=	0;
							bScrewed1							:=	TRUE;	
						END_IF
						IF tonMomentaryScrewing2Timer.Q OR bWarning2 THEN
							mcScrewer2Stop.Execute				:=	TRUE;
							bGripper2Actuator					:=	FALSE;
							mcScrewer2TorqueControl.Execute		:=	FALSE;
							uiScrewing2TorqueControl			:=	0;
							bScrewed2							:=	TRUE;		
						END_IF*)
								
						IF tonMomentaryScrewing1Timer.Q OR bWarning1 THEN
							bGripper1Actuator					:=	FALSE;
							bScrewed1							:=	TRUE;	
						END_IF
						IF tonMomentaryScrewing2Timer.Q OR bWarning2 THEN
							bGripper2Actuator					:=	FALSE;
							bScrewed2							:=	TRUE;		
						END_IF
				
						IF tonTightScrewing1TimerAndOpenedGripper.Q OR bWarning1 THEN
							mcScrewer1Stop.Execute				:=	TRUE;
							mcScrewer1TorqueControl.Execute		:=	FALSE;
						END_IF
						IF tonTightScrewing2TimerAndOpenedGripper.Q OR bWarning2 THEN
							mcScrewer2Stop.Execute				:=	TRUE;
							mcScrewer2TorqueControl.Execute		:=	FALSE;
						END_IF											
				
						// Warunki zakręcenia zaleznie od uruchomionej zakręcarki
//						IF (bScrewed1 OR NOT bRun1) AND (bScrewed2 OR NOT bRun2) AND
//							(mcScrewer1Stop.Done OR NOT mcScrewer1Stop.Execute) AND 
//							(mcScrewer2Stop.Done OR NOT mcScrewer2Stop.Execute) THEN
						IF (tonTightScrewing1TimerAndOpenedGripper.Q OR NOT bRun1) AND (tonTightScrewing2TimerAndOpenedGripper.Q OR NOT bRun2) AND
							(mcScrewer1Stop.Done OR NOT mcScrewer1Stop.Execute) AND 
							(mcScrewer2Stop.Done OR NOT mcScrewer2Stop.Execute) THEN
								mcScrewer1Stop.Execute			:= FALSE;
								mcScrewer2Stop.Execute			:= FALSE;
								iScrewingCase					:= iScrewingCase + 10;		
						END_IF
					20:
						(* Rozgearowanie osi *)
						mcHeightGearOut.Execute				:=	TRUE;
						mcHeightGearInMultiMaster.Enable	:=	FALSE;
	
						IF  mcHeightGearOut.Done THEN
							mcHeightGearOut.Execute					:= FALSE;
							eRunningState							:= E_GripperScrewer.eHolding;	
							iScrewingCase							:= 0;	
						END_IF			
					END_CASE
END_ACTION

ACTION Running6ScrewingPositionTorqueMode:
				(********* TRYB POZYCYJNY  *********)
				
				lrPackageThreadPitch;	
				(*Wymuszanie zwiększonego momentu przez 1/4 całego zakręcania*)
				IF ABS(ABS(lrStartPosition1)-ABS(Screwing1AxisRef.NcToPlc.ActPos))>(lrPackageTurnoversToFullScrewed*360.0/7)  THEN 
							uiScrewing1TorqueControl			:=	(INT_TO_UINT(iScrewer1SetTorque+3)*10)+(iScrewer1AddTorque*10);	
				ELSE		uiScrewing1TorqueControl			:=	6000;
				END_IF
				//uiScrewing1TorqueControl			:=	(INT_TO_UINT(iScrewerSetTorque+3)*10)+iScrewer1AddTorque;	
				(*Wymuszanie zwiększonego momentu przez 1/4 całego zakręcania*)
				IF ABS(ABS(lrStartPosition2)-ABS(Screwing2AxisRef.NcToPlc.ActPos))>(lrPackageTurnoversToFullScrewed*360.0/7)  THEN 
							uiScrewing2TorqueControl			:=	(INT_TO_UINT(iScrewer2SetTorque+3)*10)+(iScrewer2AddTorque*10);		
				ELSE		uiScrewing2TorqueControl			:=	6000;
				END_IF	

					CASE iScrewingCase OF 	
					0:
						(* Wersja 2 - gearowanie Multi Master***************************************************************) 
						IF iTool <> 2 THEN
							bGripper1Actuator						:=	bRun1; // Ponowne załączanie chwytaków, dlatego
							bGripper2Actuator						:=	bRun2; // że jest możliwa duża ilość opcji
						ELSE
							bGripper1Actuator						:=	FALSE; // Ponowne załączanie chwytaków, dlatego
							bGripper2Actuator						:=	FALSE; // że jest możliwa duża ilość opcji
						END_IF
						mcHeightGearInMultiMaster.Enable			:=	TRUE;				
						(* Start zakręcania *)
						IF	mcHeightGearInMultiMaster.InGear AND 
							(tonGripper1Delay.Q OR sTool = 'ksztaltowa/do kulek' OR NOT bRun1) AND (tonGripper2Delay.Q OR sTool = 'ksztaltowa/do kulek' OR NOT bRun2) // ton'y powinny być już wczesniej załączone jeżeli były chwytaki	
						THEN

							CASE iScrewing2Case OF 	
								
							0:
							
								mcScrewer1MoveVelocity2.Velocity		:=	5000;
								mcScrewer1MoveVelocity2.Execute		:=	bRun1;
								mcScrewer1MoveVelocity2.Direction	:=	MC_Positive_Direction;
																				
								mcScrewer2MoveVelocity2.Velocity		:=	5000;
								mcScrewer2MoveVelocity2.Execute		:=	bRun2;
								mcScrewer2MoveVelocity2.Direction	:=	MC_Positive_Direction;	
	
								iScrewing2Case						:=	iScrewing2Case + 10;										
							
							10:
								mcScrewer1MoveVelocity2.Execute		:=	FALSE;
								mcScrewer2MoveVelocity2.Execute		:=	FALSE;
							
								iScrewing2Case						:=	iScrewing2Case + 10;
	
							20:
							
								mcScrewer1MoveVelocity.Velocity		:=	lrScrewerSpeed;		
								mcScrewer1MoveVelocity.Direction	:=	MC_Positive_Direction;	
								IF ABS(ABS(lrStartPosition1)-ABS(Screwing1AxisRef.NcToPlc.ActPos))>(lrPackageTurnoversToFullScrewed*360.0/7)  THEN 									
									mcScrewer1MoveVelocity.Execute		:=	bRun1;									
								END_IF
								mcScrewer2MoveVelocity.Velocity		:=	lrScrewerSpeed;	
								mcScrewer1MoveVelocity.Direction		:=	MC_Positive_Direction;	
								IF ABS(ABS(lrStartPosition2)-ABS(Screwing2AxisRef.NcToPlc.ActPos))>(lrPackageTurnoversToFullScrewed*360.0/7)  THEN 
	
									mcScrewer2MoveVelocity.Execute		:=	bRun2;
								END_IF			

								IF (mcScrewer1MoveVelocity.Execute OR NOT bRun1) AND (mcScrewer2MoveVelocity.Execute OR NOT bRun2) THEN
									iScrewing2Case					:= 0	;
									iScrewingCase					:= iScrewingCase + 10;		
								END_IF
								
							END_CASE
							
						END_IF
						
					10:	
					
						(*Zmniejszanie prędkości jeżeli jest już przytrzymanie*)
						IF tonTightScrewing1Timer.ET > T#0S AND Screwing1AxisRef.NcToPlc.ActVelo < 10 THEN
							//mcScrewer1MoveVelocity.Execute		:= FALSE;
							//mcScrewer1MoveVelocity2.Execute		:= FALSE;
							
							//mcScrewer1MoveVelocity3.Velocity	:=	10;
							//mcScrewer1MoveVelocity3.Execute		:=	bRun1;
							//mcScrewer1MoveVelocity3.Direction	:=	MC_Positive_Direction;		

							rScrewing1ProportionalGain	:= 0;
							//rScrewing2ProportionalGain	:= 0;												
						END_IF
						
						IF tonTightScrewing2Timer.ET > T#0S AND Screwing2AxisRef.NcToPlc.ActVelo < 10 THEN
							//mcScrewer2MoveVelocity.Execute		:= FALSE;
							//mcScrewer2MoveVelocity2.Execute		:= FALSE;
							
							//mcScrewer2MoveVelocity3.Velocity	:=	10;
							//mcScrewer2MoveVelocity3.Execute		:=	bRun1;
							//mcScrewer2MoveVelocity3.Direction	:=	MC_Positive_Direction;		

							//rScrewing1ProportionalGain	:= 0;
							rScrewing2ProportionalGain	:= 0;												
						END_IF					
					
						(* Sprawdzanie czy osiągnięto moment lub zbyt długie zakracanie*)				
						IF tonTightScrewing1Timer.Q OR bWarning1 THEN
							bGripper1Actuator					:=	FALSE;
							bScrewed1							:=	TRUE;	
						END_IF
						IF tonTightScrewing2Timer.Q OR bWarning2 THEN
							bGripper2Actuator					:=	FALSE;
							bScrewed2							:=	TRUE;		
						END_IF
	
						IF tonTightScrewing1TimerAndOpenedGripper.Q THEN
							mcScrewer1Stop.Execute				:=	TRUE;
							mcScrewer1MoveVelocity.Execute		:=	FALSE;
							mcScrewer1MoveVelocity2.Execute		:=	FALSE;
							mcScrewer1MoveVelocity3.Execute		:=	FALSE;							
							uiScrewing1TorqueControl			:=	0;
						END_IF
						IF tonTightScrewing2TimerAndOpenedGripper.Q THEN
							mcScrewer2Stop.Execute				:=	TRUE;
							mcScrewer2MoveVelocity.Execute		:=	FALSE;
							mcScrewer2MoveVelocity2.Execute		:=	FALSE;	
							mcScrewer2MoveVelocity3.Execute		:=	FALSE;							
							uiScrewing2TorqueControl			:=	0;
						END_IF
					
						// Warunki zakręcenia zaleznie od uruchomionej zakręcarki
						IF (tonTightScrewing1TimerAndOpenedGripper.Q OR NOT bRun1) AND (tonTightScrewing2TimerAndOpenedGripper.Q OR NOT bRun2) AND
							(mcScrewer1Stop.Done OR NOT mcScrewer1Stop.Execute) AND 
							(mcScrewer2Stop.Done OR NOT mcScrewer2Stop.Execute) THEN
								mcScrewer1Stop.Execute			:= FALSE;
								mcScrewer2Stop.Execute			:= FALSE;
								iScrewingCase					:= iScrewingCase + 10;		
						END_IF
						
					20:
						(* Rozgearowanie osi *)
						mcHeightGearOut.Execute				:=	TRUE;
						mcHeightGearInMultiMaster.Enable	:=	FALSE;
	
						IF  mcHeightGearOut.Done THEN
							mcHeightGearOut.Execute					:= FALSE;
							eRunningState							:= E_GripperScrewer.eHolding;	
							iScrewingCase							:= 0;	
						END_IF			
					END_CASE
END_ACTION

ACTION Screwer1ControlBlocks:
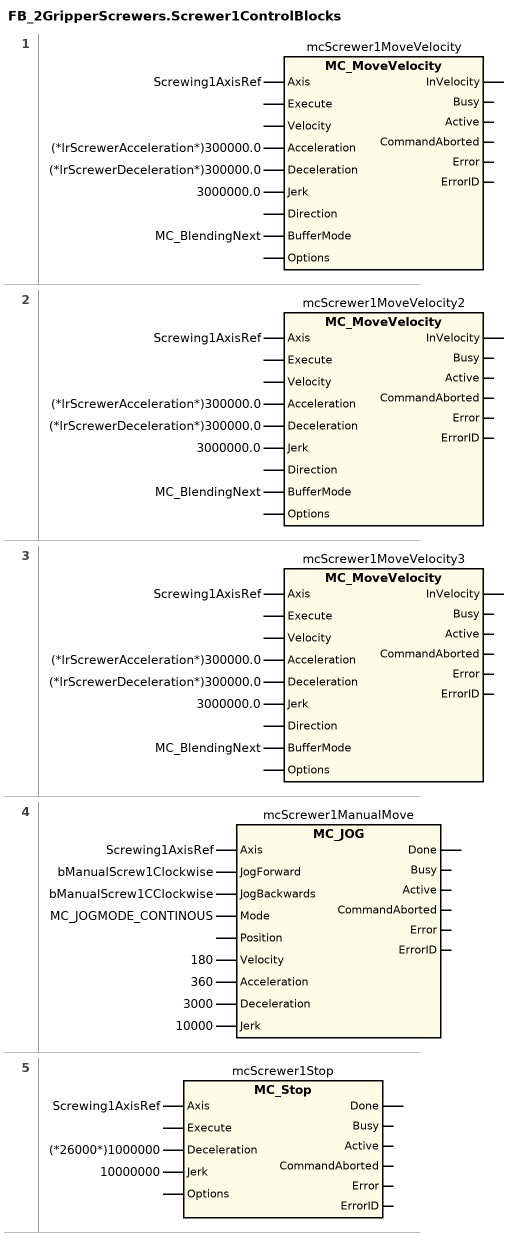
// NETWORK 1
mcScrewer1MoveVelocity(
    Axis := Screwing1AxisRef,
    Acceleration := (*lrScrewerAcceleration*)300000.0,
    Deceleration := (*lrScrewerDeceleration*)300000.0,
    Jerk := 3000000.0,
    BufferMode := MC_BlendingNext); // MC_MoveVelocity

// NETWORK 2
mcScrewer1MoveVelocity2(
    Axis := Screwing1AxisRef,
    Acceleration := (*lrScrewerAcceleration*)300000.0,
    Deceleration := (*lrScrewerDeceleration*)300000.0,
    Jerk := 3000000.0,
    BufferMode := MC_BlendingNext); // MC_MoveVelocity

// NETWORK 3
mcScrewer1MoveVelocity3(
    Axis := Screwing1AxisRef,
    Acceleration := (*lrScrewerAcceleration*)300000.0,
    Deceleration := (*lrScrewerDeceleration*)300000.0,
    Jerk := 3000000.0,
    BufferMode := MC_BlendingNext); // MC_MoveVelocity

// NETWORK 4
mcScrewer1ManualMove(
    Axis := Screwing1AxisRef,
    JogForward := bManualScrew1Clockwise,
    JogBackwards := bManualScrew1CClockwise,
    Mode := MC_JOGMODE_CONTINOUS,
    Velocity := 180,
    Acceleration := 360,
    Deceleration := 3000,
    Jerk := 10000); // MC_JOG

// NETWORK 5
mcScrewer1Stop(Axis := Screwing1AxisRef, Deceleration := (*26000*)1000000, Jerk := 10000000); // MC_Stop

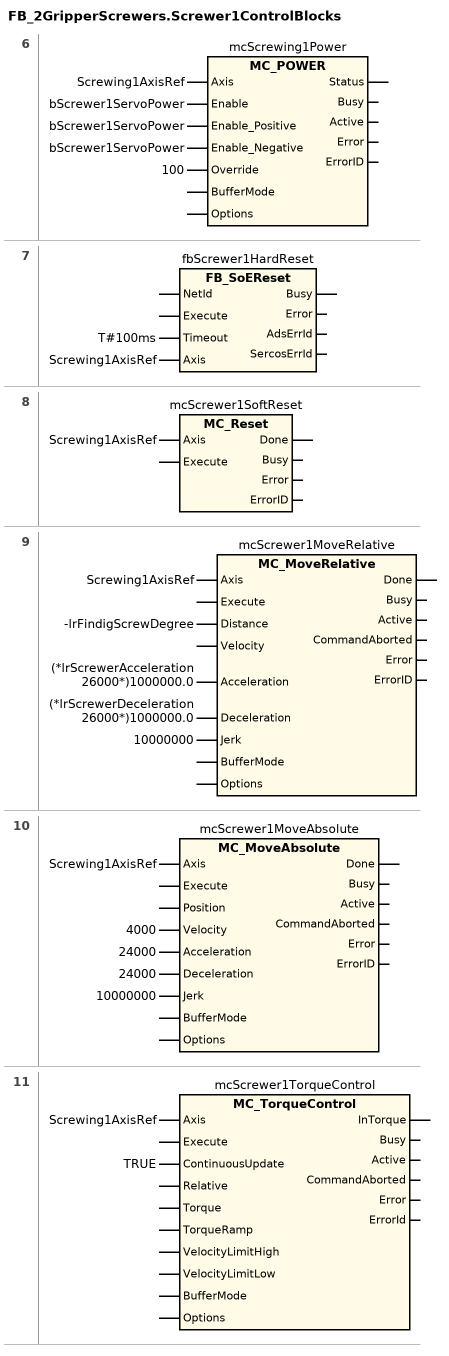
// NETWORK 6
mcScrewing1Power(
    Axis := Screwing1AxisRef,
    Enable := bScrewer1ServoPower,
    Enable_Positive := bScrewer1ServoPower,
    Enable_Negative := bScrewer1ServoPower,
    Override := 100); // MC_POWER

// NETWORK 7
fbScrewer1HardReset(Timeout := T#100ms, Axis := Screwing1AxisRef); // FB_SoEReset

// NETWORK 8
mcScrewer1SoftReset(Axis := Screwing1AxisRef); // MC_Reset

// NETWORK 9
mcScrewer1MoveRelative(
    Axis := Screwing1AxisRef,
    Distance := -lrFindigScrewDegree,
    Acceleration := (*lrScrewerAcceleration 26000*)1000000.0,
    Deceleration := (*lrScrewerDeceleration 26000*)1000000.0,
    Jerk := 10000000); // MC_MoveRelative

// NETWORK 10
mcScrewer1MoveAbsolute(
    Axis := Screwing1AxisRef,
    Velocity := 4000,
    Acceleration := 24000,
    Deceleration := 24000,
    Jerk := 10000000); // MC_MoveAbsolute

// NETWORK 11
mcScrewer1TorqueControl(Axis := Screwing1AxisRef, ContinuousUpdate := TRUE); // MC_TorqueControl

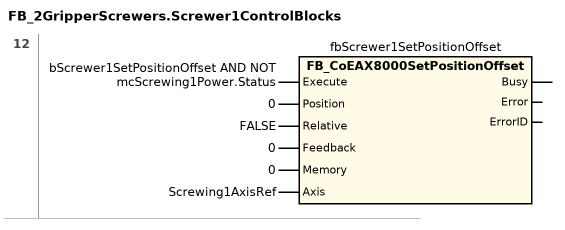
// NETWORK 12
fbScrewer1SetPositionOffset(
    Execute := bScrewer1SetPositionOffset AND NOT mcScrewing1Power.Status,
    Position := 0,
    Relative := FALSE,
    Feedback := 0,
    Memory := 0,
    Axis := Screwing1AxisRef); // FB_CoEAX8000SetPositionOffset
END_ACTION

ACTION Screwer2ControlBlocks:
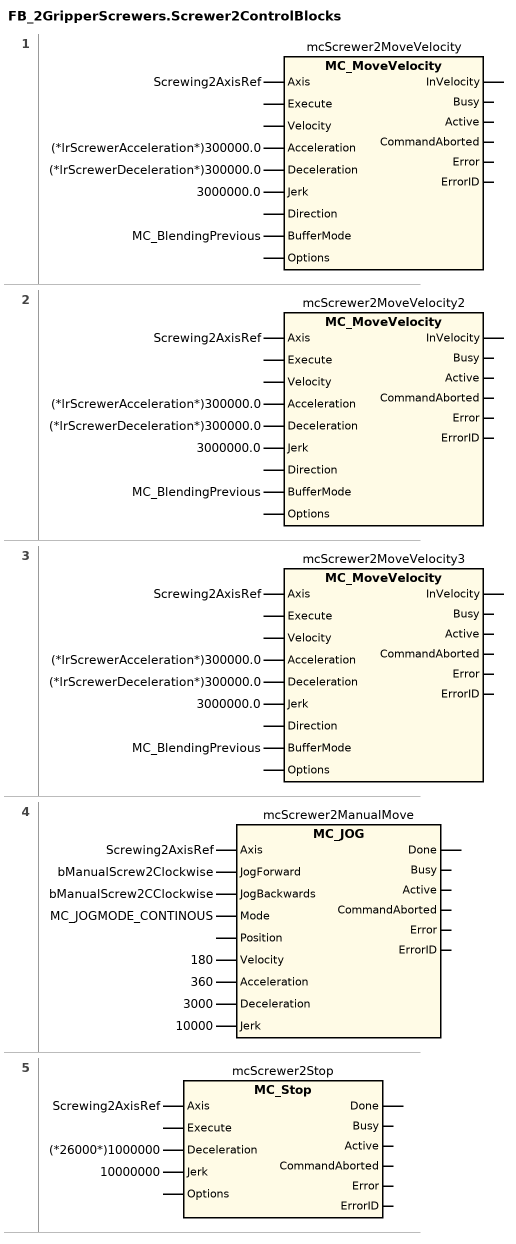
// NETWORK 1
mcScrewer2MoveVelocity(
    Axis := Screwing2AxisRef,
    Acceleration := (*lrScrewerAcceleration*)300000.0,
    Deceleration := (*lrScrewerDeceleration*)300000.0,
    Jerk := 3000000.0,
    BufferMode := MC_BlendingPrevious); // MC_MoveVelocity

// NETWORK 2
mcScrewer2MoveVelocity2(
    Axis := Screwing2AxisRef,
    Acceleration := (*lrScrewerAcceleration*)300000.0,
    Deceleration := (*lrScrewerDeceleration*)300000.0,
    Jerk := 3000000.0,
    BufferMode := MC_BlendingPrevious); // MC_MoveVelocity

// NETWORK 3
mcScrewer2MoveVelocity3(
    Axis := Screwing2AxisRef,
    Acceleration := (*lrScrewerAcceleration*)300000.0,
    Deceleration := (*lrScrewerDeceleration*)300000.0,
    Jerk := 3000000.0,
    BufferMode := MC_BlendingPrevious); // MC_MoveVelocity

// NETWORK 4
mcScrewer2ManualMove(
    Axis := Screwing2AxisRef,
    JogForward := bManualScrew2Clockwise,
    JogBackwards := bManualScrew2CClockwise,
    Mode := MC_JOGMODE_CONTINOUS,
    Velocity := 180,
    Acceleration := 360,
    Deceleration := 3000,
    Jerk := 10000); // MC_JOG

// NETWORK 5
mcScrewer2Stop(Axis := Screwing2AxisRef, Deceleration := (*26000*)1000000, Jerk := 10000000); // MC_Stop

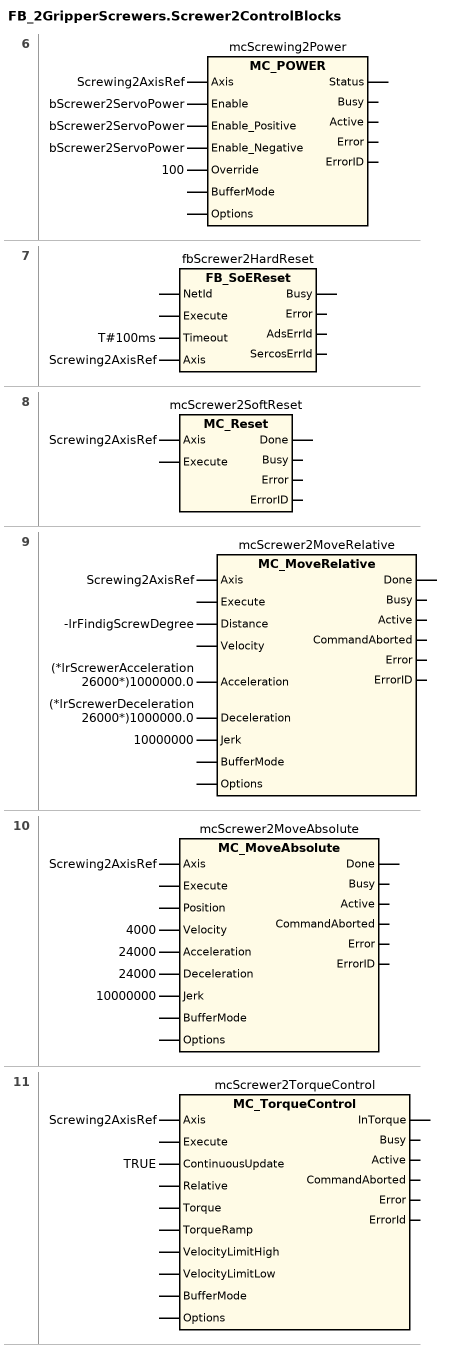
// NETWORK 6
mcScrewing2Power(
    Axis := Screwing2AxisRef,
    Enable := bScrewer2ServoPower,
    Enable_Positive := bScrewer2ServoPower,
    Enable_Negative := bScrewer2ServoPower,
    Override := 100); // MC_POWER

// NETWORK 7
fbScrewer2HardReset(Timeout := T#100ms, Axis := Screwing2AxisRef); // FB_SoEReset

// NETWORK 8
mcScrewer2SoftReset(Axis := Screwing2AxisRef); // MC_Reset

// NETWORK 9
mcScrewer2MoveRelative(
    Axis := Screwing2AxisRef,
    Distance := -lrFindigScrewDegree,
    Acceleration := (*lrScrewerAcceleration 26000*)1000000.0,
    Deceleration := (*lrScrewerDeceleration 26000*)1000000.0,
    Jerk := 10000000); // MC_MoveRelative

// NETWORK 10
mcScrewer2MoveAbsolute(
    Axis := Screwing2AxisRef,
    Velocity := 4000,
    Acceleration := 24000,
    Deceleration := 24000,
    Jerk := 10000000); // MC_MoveAbsolute

// NETWORK 11
mcScrewer2TorqueControl(Axis := Screwing2AxisRef, ContinuousUpdate := TRUE); // MC_TorqueControl

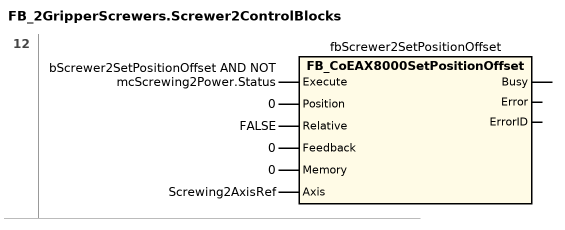
// NETWORK 12
fbScrewer2SetPositionOffset(
    Execute := bScrewer2SetPositionOffset AND NOT mcScrewing2Power.Status,
    Position := 0,
    Relative := FALSE,
    Feedback := 0,
    Memory := 0,
    Axis := Screwing2AxisRef); // FB_CoEAX8000SetPositionOffset
END_ACTION

ACTION Simulation:
(* Przyśpieszanie bloku gdy jest włączona symulacja*)

//tonSimulationScrewing1			(IN:=eRunningState=E_GripperScrewer.eScrewing 	AND bRun1 AND NOT bScrewed1 AND bSimulation,	PT:=T#0MS);
//tonSimulationScrewing2			(IN:=eRunningState=E_GripperScrewer.eScrewing 	AND bRun1 AND NOT bScrewed2 AND bSimulation,	PT:=T#0MS);

IF bSimulation THEN 			// Włączona symulacja
	tTooLongScrewing1 := T#250MS;
	tTooLongScrewing2 := T#250MS;	
ELSE							// Normalna praca
	tTooLongScrewing1 := T#3S; 	//Zmienić na 2
	tTooLongScrewing2 := T#3S;	//Zmienić na 2
END_IF
END_ACTION

ACTION Statistics:

IF LREAL_TO_INT(lrHeightEndScrewingPosition)<> LREAL_TO_INT(lrHeightReadyPosition) THEN
	rtrigCycleTimerRead(CLK:=LREAL_TO_INT(lrHeightActualPosition) = LREAL_TO_INT(lrHeightReadyPosition));
	IF rtrigCycleTimerRead.Q THEN
			tCycleTime:=tonCycleTimer.ET;
	END_IF
	tonCycleTimer(IN:=LREAL_TO_INT(lrHeightActualPosition) <> LREAL_TO_INT(lrHeightReadyPosition),PT:=T#1D);	
ELSE
	rtrigCycleTimerRead(CLK:=(eRunningState=E_GripperScrewer.eDone) OR (eRunningState=E_GripperScrewer.eNotDone));
	IF rtrigCycleTimerRead.Q THEN
		tCycleTime:=tonCycleTimer.ET;
	END_IF
	tonCycleTimer(IN:=eRunningState>E_GripperScrewer.eReady,PT:=T#1D);
END_IF
END_ACTION

ACTION Tools:
(*Narzędzia*)
AsToolDescription[0] := 'Głowica dwuszczękowa';
AsToolDescription[1] := 'Głowica trójszczękowa'; 
AsToolDescription[2] := 'Głowica kształtowa/do kulek';
AsToolDescription[3] := 'Głowica wbijająca'; 
AsToolDescription[4] := 'Głowica zasysająca';


(*Głowica wbijająca*)
IF iTool = 3 THEN
	bOptionCapPushingWithoutScrewing := TRUE;
ELSE
	bOptionCapPushingWithoutScrewing := FALSE;
END_IF

(*Przepisanie wybranego narzędzia do zmiennej typu string*)
(*!!!!! NIE ZMIENIAĆ OPISÓW, POWIĄZANE W PROGRAMIE !!!!!!*)
(* Wysokość narzędzia od pkt. bazowania

		Glowica dwuszczekowa
           |	|
		   |	|
	|------|    |-----|
	|	 _______	  |
	|	|		  |   |
   ||	||		  |   |
   ||	||		  |	  |
   |---- |		  -----	<-pkt. bazowania 	<-|
   |	 |	                                  |
   |	 ---|	  							iToolHeight (mm)
   |druk	|                                 |
   ---------|	  							<-|

*)


IF iTool = 0 THEN sTool := 'dwuszczekowa';			iToolHeight	:=	23;		END_IF 
IF iTool = 1 THEN sTool := 'trojszczekowa';			iToolHeight	:=	-5;	END_IF 
IF iTool = 2 THEN sTool := 'ksztaltowa/do kulek';	iToolHeight	:=	-5;		END_IF 
IF iTool = 3 THEN sTool := 'wbijajaca';				iToolHeight	:=	23;		END_IF 
IF iTool = 4 THEN sTool := 'zasysajaca';			iToolHeight	:=	-4;		END_IF
END_ACTION

ACTION TorqueControl:

(*Konfiguracja MC_TorqueControl*)
//T_TorqueControlOptions;
mcScrewer1TorqueControl.Options.EnableManualTorqueStartValue := TRUE;
mcScrewer1TorqueControl.Options.ManualTorqueStartValue       := Screwing1AxisRef.NcToPlc.ActTorque;

mcScrewer2TorqueControl.Options.EnableManualTorqueStartValue := TRUE;
mcScrewer2TorqueControl.Options.ManualTorqueStartValue       :=  Screwing2AxisRef.NcToPlc.ActTorque;
END_ACTION

ACTION Warnings:
//Resetowanie warningów przy nastepnym cyklu

IF rtRun1.Q  OR rtRun2.Q THEN
	
	bWarning1			:=	FALSE;
	bWarning1A			:=	FALSE;
	bWarning1B			:=	FALSE;
	bWarning1C			:=	FALSE;
	bWarning1D			:=	FALSE;
	bWarning1E			:=	FALSE;	
	bWarning2			:=	FALSE;
	bWarning2A			:=	FALSE;
	bWarning2B			:=	FALSE;
	bWarning2C			:=	FALSE;
	bWarning2D			:=	FALSE;
	bWarning2E			:=	FALSE;
END_IF
END_ACTION

END_FUNCTION_BLOCK

(* stored: Version 1.1.0.1, ProductVersion 3.1.4026.13, FileIdentifier 963fe0be0f0aefc7d55b05f7ee3b4490068b601f, FileSignature 16285db06acca9e8f7652178182512c3840cad131fa7eafdd5a5707dc4eeeaad08ec5ff2682d44b888650e57d45b4eb0ab397fa5fd33f0d03affc2fe1e1f1c3cb8bd306fd82cace553e3862c288b85a8e49ff9c54bd2d986f324c5c5683a02e5d1279a682130870875218b9925ddda6daaab42f8f938e598f66b54964b4ace55b6528d557ac851be7eec1f1fd0c1ea310fe13ff503b6b52f29d96c1a3d6ece07e2039e67fd9e23f428b0c5f5262e30b6565caa13c4beb48b7772c18eebd388ac5d569b2e47b231af0cc912dcdc909047a00f5ee9c37d004bf96e92566f1d7d6372f3a40e4675061ef719205ce295a2a3d8f40ff8080d7ada2d4d44cb68108776
   POU FB_2GripperScrewers: Id {2e6dda3d-a09e-43dc-83d8-5b983083272b}, SpecialFunc None
   Folder Methods: Id {dc88b3ef-0515-4453-9b81-4aa6aca1eb6e}
   Action AdjustingTorque: Id {b7cf1dd4-e1d2-4859-812e-43c1eee05297}
   Action aStationID: Id {40121b5c-09a5-49ba-b644-6b8488e917ce}
   Action aTesty: Id {0c08d85b-f8b5-4fa1-b6f1-411521ca0034}
   Action Control: Id {b3209faf-d460-4f3f-a56b-dd9d3de3e0ec}
   Action ErrorHandling: Id {fe0c8aa6-99ff-497a-b6b0-8082ea45ddeb}
   Action HeightControlBlocks: Id {566db1c7-3709-48eb-a407-a42673ab463a}
   Action Homing: Id {fece0f5f-43f4-415c-bb30-b2c92e38c294}
   Action Limits: Id {33fd4837-7b88-4191-b1a5-61222e49d220}
   Method M_PrepareToReady: Id {42205c1d-fc2f-4cde-8fd8-486a0aafef30}
   Action ManualMovements: Id {2359265d-3084-42e6-9a0d-0fac2b55009d}
   Action ManualMovementsStepMode: Id {18057dd4-187d-4a2e-b906-4af4374f8fd8}
   Action ReadScrewingTorque: Id {37f8e9c2-9f74-40bb-a650-dd7834c6b2f1}
   Action ResetCommands: Id {4186105b-87be-4434-830c-f14521986b42}
   Action Running: Id {483d300e-118d-4df7-b978-ada62a1e7d7d}
   Action Running2ToPushingPosition: Id {fd83140c-dd59-4891-a724-065ef3f0a097}
   Action Running5FindingScrew: Id {17b75710-8931-4d58-a841-31199963f3c9}
   Action Running6ScrewingMomentaryMode: Id {6d6ccd6b-73db-4738-a076-05023edf7e63}
   Action Running6ScrewingPositionTorqueMode: Id {b9a3ffb1-0c1a-4a9b-8c65-066c02efd576}
   Action Screwer1ControlBlocks: Id {32b09e26-fe16-4d56-932e-347d3814014b}
   Action Screwer2ControlBlocks: Id {f6131b1b-2e49-43b1-a5e2-8c99fbe6342c}
   Action Simulation: Id {cf861b4b-d26f-4ecc-b25e-480c8a95740e}
   Action Statistics: Id {c39965e8-4b50-4276-b3cf-9906d5a315d2}
   Action Tools: Id {c1f3f0fa-96c6-4030-b793-e67f94617304}
   Action TorqueControl: Id {8eed6ea9-13e0-4f1a-8680-2d0ebd6c9b8c}
   Action Warnings: Id {9de86b7c-d076-44e9-ae89-87418569aad2} *)
